// TIA Portal V20 export
TYPE "LKinCtrl_typeDynamics"
   STRUCT
      path : "LKinCtrl_typePathDynamics";   // Specification of the path dynamics
      orientation : "LKinCtrl_typePathDynamics";   // Specification of the orientation dynamics
      dynamicAdaption : DInt := 1;   // 0=no dynamic adaption, 1=dynamic adaptation with segmentation of the path, 2=dynamic adaptation without segmentation of the path
      directionA : DInt := 3;   // 1=positive direction, 2=negative direction, 3=shortest distance
      sPTP : "LKinCtrl_typeSPTPDynamics";   // Specification of the dynamic factor for sptp movement
   END_STRUCT;
END_TYPE
